// TIA Portal V20 export
DATA_BLOCK "DB_NcVarSelect_MA_JOG_VELO_RAPID"   // DB65
{ S7_Optimized_Access := 'TRUE' }
// stored: MemoryReserve 100
   VAR
      "$MA_JOG_VELO_RAPID_Axis01_X" { S7_SetPoint := 'True'} : "LBP_typeNCVariableTokenLReal";
      "$MA_JOG_VELO_RAPID_Axis02_Y" { S7_SetPoint := 'True'} : "LBP_typeNCVariableTokenLReal";
      "$MA_JOG_VELO_RAPID_Axis03_ZM" { S7_SetPoint := 'True'} : "LBP_typeNCVariableTokenLReal";
      "$MA_JOG_VELO_RAPID_Axis04_B" { S7_SetPoint := 'True'} : "LBP_typeNCVariableTokenLReal";
      "$MA_JOG_VELO_RAPID_Axis05_U1" { S7_SetPoint := 'True'} : "LBP_typeNCVariableTokenLReal";
      "$MA_JOG_VELO_RAPID_Axis06_U2" { S7_SetPoint := 'True'} : "LBP_typeNCVariableTokenLReal";
      "$MA_JOG_VELO_RAPID_Axis07_V" { S7_SetPoint := 'True'} : "LBP_typeNCVariableTokenLReal";
      "$MA_JOG_VELO_RAPID_Axis08_W" { S7_SetPoint := 'True'} : "LBP_typeNCVariableTokenLReal";
      "$MA_JOG_VELO_RAPID_Axis09_ZL" { S7_SetPoint := 'True'} : "LBP_typeNCVariableTokenLReal";
   END_VAR
BEGIN
   "$MA_JOG_VELO_RAPID_Axis01_X".token.syntaxId := 16#82;
   "$MA_JOG_VELO_RAPID_Axis01_X".token.areaAndUnit := 16#61;
   "$MA_JOG_VELO_RAPID_Axis01_X".token.column := 16#7D0A;
   "$MA_JOG_VELO_RAPID_Axis01_X".token.row := 16#1;
   "$MA_JOG_VELO_RAPID_Axis01_X".token.blockType := 16#1A;
   "$MA_JOG_VELO_RAPID_Axis01_X".token.numberOfRows := 16#1;
   "$MA_JOG_VELO_RAPID_Axis01_X".token.dataTypeCode := 16#F;
   "$MA_JOG_VELO_RAPID_Axis01_X".token.length := 16#8;
   "$MA_JOG_VELO_RAPID_Axis02_Y".token.syntaxId := 16#82;
   "$MA_JOG_VELO_RAPID_Axis02_Y".token.areaAndUnit := 16#62;
   "$MA_JOG_VELO_RAPID_Axis02_Y".token.column := 16#7D0A;
   "$MA_JOG_VELO_RAPID_Axis02_Y".token.row := 16#1;
   "$MA_JOG_VELO_RAPID_Axis02_Y".token.blockType := 16#1A;
   "$MA_JOG_VELO_RAPID_Axis02_Y".token.numberOfRows := 16#1;
   "$MA_JOG_VELO_RAPID_Axis02_Y".token.dataTypeCode := 16#F;
   "$MA_JOG_VELO_RAPID_Axis02_Y".token.length := 16#8;
   "$MA_JOG_VELO_RAPID_Axis03_ZM".token.syntaxId := 16#82;
   "$MA_JOG_VELO_RAPID_Axis03_ZM".token.areaAndUnit := 16#63;
   "$MA_JOG_VELO_RAPID_Axis03_ZM".token.column := 16#7D0A;
   "$MA_JOG_VELO_RAPID_Axis03_ZM".token.row := 16#1;
   "$MA_JOG_VELO_RAPID_Axis03_ZM".token.blockType := 16#1A;
   "$MA_JOG_VELO_RAPID_Axis03_ZM".token.numberOfRows := 16#1;
   "$MA_JOG_VELO_RAPID_Axis03_ZM".token.dataTypeCode := 16#F;
   "$MA_JOG_VELO_RAPID_Axis03_ZM".token.length := 16#8;
   "$MA_JOG_VELO_RAPID_Axis04_B".token.syntaxId := 16#82;
   "$MA_JOG_VELO_RAPID_Axis04_B".token.areaAndUnit := 16#64;
   "$MA_JOG_VELO_RAPID_Axis04_B".token.column := 16#7D0A;
   "$MA_JOG_VELO_RAPID_Axis04_B".token.row := 16#1;
   "$MA_JOG_VELO_RAPID_Axis04_B".token.blockType := 16#1A;
   "$MA_JOG_VELO_RAPID_Axis04_B".token.numberOfRows := 16#1;
   "$MA_JOG_VELO_RAPID_Axis04_B".token.dataTypeCode := 16#F;
   "$MA_JOG_VELO_RAPID_Axis04_B".token.length := 16#8;
   "$MA_JOG_VELO_RAPID_Axis05_U1".token.syntaxId := 16#82;
   "$MA_JOG_VELO_RAPID_Axis05_U1".token.areaAndUnit := 16#65;
   "$MA_JOG_VELO_RAPID_Axis05_U1".token.column := 16#7D0A;
   "$MA_JOG_VELO_RAPID_Axis05_U1".token.row := 16#1;
   "$MA_JOG_VELO_RAPID_Axis05_U1".token.blockType := 16#1A;
   "$MA_JOG_VELO_RAPID_Axis05_U1".token.numberOfRows := 16#1;
   "$MA_JOG_VELO_RAPID_Axis05_U1".token.dataTypeCode := 16#F;
   "$MA_JOG_VELO_RAPID_Axis05_U1".token.length := 16#8;
   "$MA_JOG_VELO_RAPID_Axis06_U2".token.syntaxId := 16#82;
   "$MA_JOG_VELO_RAPID_Axis06_U2".token.areaAndUnit := 16#66;
   "$MA_JOG_VELO_RAPID_Axis06_U2".token.column := 16#7D0A;
   "$MA_JOG_VELO_RAPID_Axis06_U2".token.row := 16#1;
   "$MA_JOG_VELO_RAPID_Axis06_U2".token.blockType := 16#1A;
   "$MA_JOG_VELO_RAPID_Axis06_U2".token.numberOfRows := 16#1;
   "$MA_JOG_VELO_RAPID_Axis06_U2".token.dataTypeCode := 16#F;
   "$MA_JOG_VELO_RAPID_Axis06_U2".token.length := 16#8;
   "$MA_JOG_VELO_RAPID_Axis07_V".token.syntaxId := 16#82;
   "$MA_JOG_VELO_RAPID_Axis07_V".token.areaAndUnit := 16#67;
   "$MA_JOG_VELO_RAPID_Axis07_V".token.column := 16#7D0A;
   "$MA_JOG_VELO_RAPID_Axis07_V".token.row := 16#1;
   "$MA_JOG_VELO_RAPID_Axis07_V".token.blockType := 16#1A;
   "$MA_JOG_VELO_RAPID_Axis07_V".token.numberOfRows := 16#1;
   "$MA_JOG_VELO_RAPID_Axis07_V".token.dataTypeCode := 16#F;
   "$MA_JOG_VELO_RAPID_Axis07_V".token.length := 16#8;
   "$MA_JOG_VELO_RAPID_Axis08_W".token.syntaxId := 16#82;
   "$MA_JOG_VELO_RAPID_Axis08_W".token.areaAndUnit := 16#68;
   "$MA_JOG_VELO_RAPID_Axis08_W".token.column := 16#7D0A;
   "$MA_JOG_VELO_RAPID_Axis08_W".token.row := 16#1;
   "$MA_JOG_VELO_RAPID_Axis08_W".token.blockType := 16#1A;
   "$MA_JOG_VELO_RAPID_Axis08_W".token.numberOfRows := 16#1;
   "$MA_JOG_VELO_RAPID_Axis08_W".token.dataTypeCode := 16#F;
   "$MA_JOG_VELO_RAPID_Axis08_W".token.length := 16#8;
   "$MA_JOG_VELO_RAPID_Axis09_ZL".token.syntaxId := 16#82;
   "$MA_JOG_VELO_RAPID_Axis09_ZL".token.areaAndUnit := 16#69;
   "$MA_JOG_VELO_RAPID_Axis09_ZL".token.column := 16#7D0A;
   "$MA_JOG_VELO_RAPID_Axis09_ZL".token.row := 16#1;
   "$MA_JOG_VELO_RAPID_Axis09_ZL".token.blockType := 16#1A;
   "$MA_JOG_VELO_RAPID_Axis09_ZL".token.numberOfRows := 16#1;
   "$MA_JOG_VELO_RAPID_Axis09_ZL".token.dataTypeCode := 16#F;
   "$MA_JOG_VELO_RAPID_Axis09_ZL".token.length := 16#8;
END_DATA_BLOCK
